(*
	RJM Maszyny sp. z o.o.
	autor 	: Rafał Osajda
	data	: 02.02.2024
	TC		: 3.1 4024.54
	wersja	: 0.0.1.0	: pełna obsługa

	Obsługa elektrozaworu NC
*)
FUNCTION_BLOCK FB_IOElectrovalve_3on2_NC EXTENDS FB_IOElectrovalve
VAR
END_VAR

(*
	RJM Maszyny sp. z o.o.
	autor 	: Rafał Osajda
	data	: 21.02.2024
	TC		: 3.1 4024.54
	wersja	: 0.0.1.0	: pełna obsługa

	Ustawienie odpowiednich wyjść
*)METHOD Contol : BOOL
VAR_INPUT
	eAction	: E_IOElectrovalveAction;
END_VAR
CASE eAction OF
	E_IOElectrovalveAction.e_EV_Out4_Deactive	:
		bCoilA								:= FALSE;
	E_IOElectrovalveAction.e_EV_OUT4_Active	:
		bCoilA								:= TRUE;
	E_IOElectrovalveAction.e_EV_Reset			:
		bCoilA								:= FALSE;

END_CASE
bCoilB										:= FALSE;
END_METHOD

METHOD FB_init : BOOL
VAR_INPUT
	bInitRetains : BOOL; // if TRUE, the retain variables are initialized (warm start / cold start)
	bInCopyCode : BOOL;  // if TRUE, the instance afterwards gets moved into the copy code (online change)
END_VAR
THIS^.eType			:= E_IOElectrovalveType.NC_3na2;
END_METHOD

END_FUNCTION_BLOCK

(* stored: Version 1.1.0.1
   POU FB_IOElectrovalve_3on2_NC: Id {e1fe4a24-7ba7-0005-0692-39233080fb8f}, SpecialFunc None
   Method Contol: Id {9f30d02f-6ea1-07c1-2a7a-8305c2395ece}
   Method FB_init: Id {79c83901-52d6-46ac-9b2f-535d6aff250b} *)
